// TIA Portal V18 export
ORGANIZATION_BLOCK "00-Alarms"   // OB126, LAD, ProgramCycle
TITLE = Alarms / "Main Program Sweep (Cycle)"
{ S7_Optimized_Access := 'TRUE' }
VERSION : 0.1
// stored: AutoNumber true, IsIECCheckEnabled false, SetENOAutomatically false
   VAR_INPUT
      Initial_Call : Bool;   // Initial call of this OB
      Remanence : Bool;   // =True, if remanent data are available
   END_VAR
BEGIN

REGION Network 1
   // Sınıflandıramadığım Alarm Listesi
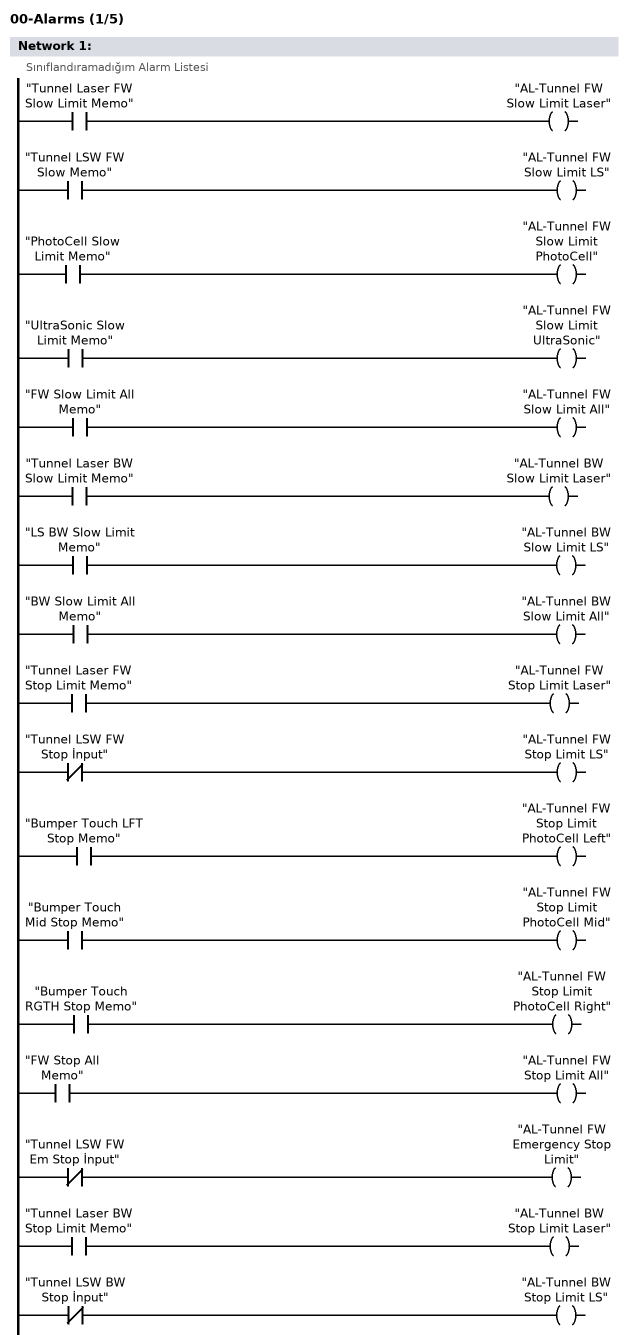
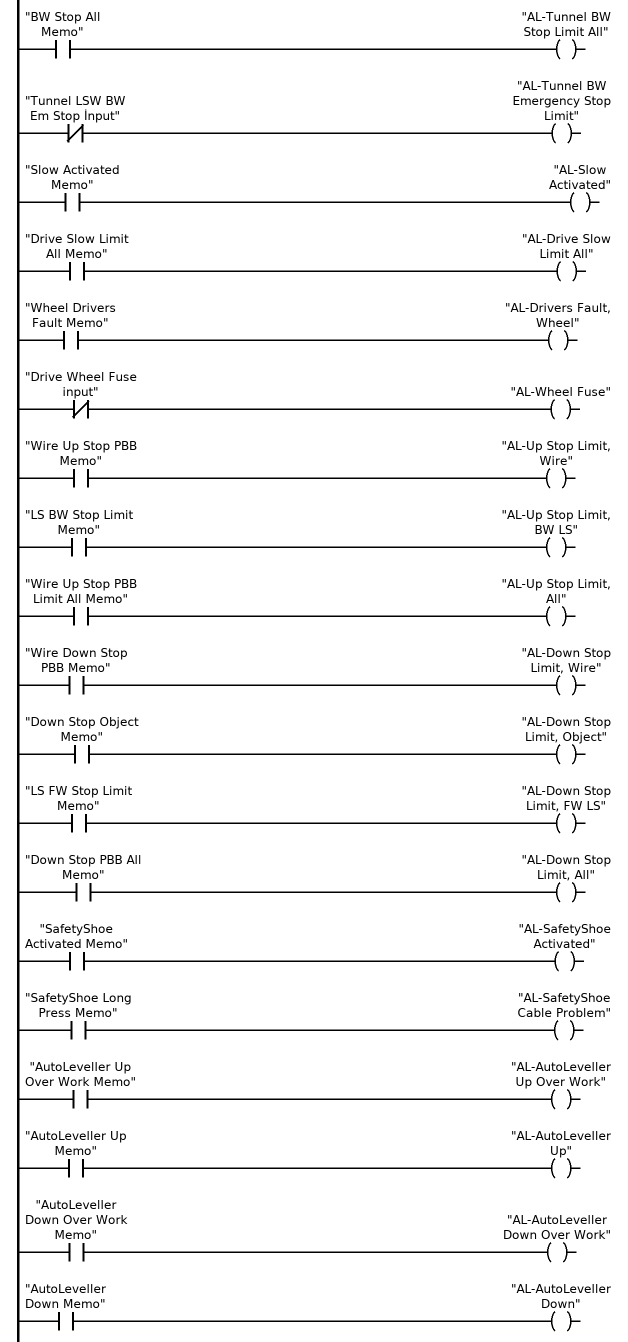
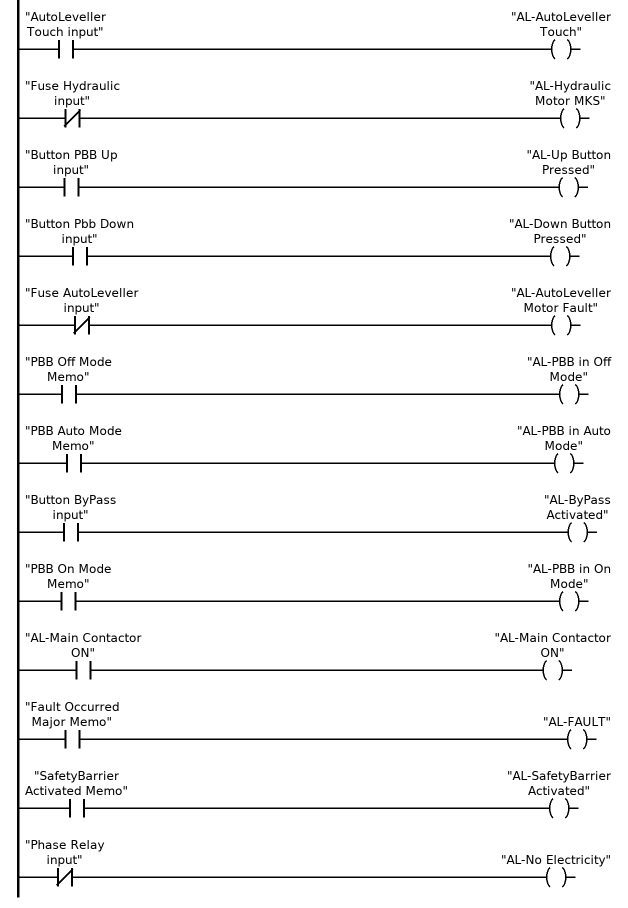
   RUNG wire#powerrail
      Contact( "Tunnel Laser FW Slow Limit Memo" )
      Coil( "AL-Tunnel FW Slow Limit Laser" )
   END_RUNG
   RUNG wire#powerrail
      Contact( "Tunnel LSW FW Slow Memo" )
      Coil( "AL-Tunnel FW Slow Limit LS" )
   END_RUNG
   RUNG wire#powerrail
      Contact( "PhotoCell Slow Limit Memo" )
      Coil( "AL-Tunnel FW Slow Limit PhotoCell" )
   END_RUNG
   RUNG wire#powerrail
      Contact( "UltraSonic Slow Limit Memo" )
      Coil( "AL-Tunnel FW Slow Limit UltraSonic" )
   END_RUNG
   RUNG wire#powerrail
      Contact( "FW Slow Limit All Memo" )
      Coil( "AL-Tunnel FW Slow Limit All" )
   END_RUNG
   RUNG wire#powerrail
      Contact( "Tunnel Laser BW Slow Limit Memo" )
      Coil( "AL-Tunnel BW Slow Limit Laser" )
   END_RUNG
   RUNG wire#powerrail
      Contact( "LS BW Slow Limit Memo" )
      Coil( "AL-Tunnel BW Slow Limit LS" )
   END_RUNG
   RUNG wire#powerrail
      Contact( "BW Slow Limit All Memo" )
      Coil( "AL-Tunnel BW Slow Limit All" )
   END_RUNG
   RUNG wire#powerrail
      Contact( "Tunnel Laser FW Stop Limit Memo" )
      Coil( "AL-Tunnel FW Stop Limit Laser" )
   END_RUNG
   RUNG wire#powerrail
      I_Contact( "Tunnel LSW FW Stop İnput" )
      Coil( "AL-Tunnel FW Stop Limit LS" )
   END_RUNG
   RUNG wire#powerrail
      Contact( "Bumper Touch LFT Stop Memo" )
      Coil( "AL-Tunnel FW Stop Limit PhotoCell Left" )
   END_RUNG
   RUNG wire#powerrail
      Contact( "Bumper Touch Mid Stop Memo" )
      Coil( "AL-Tunnel FW Stop Limit PhotoCell Mid" )
   END_RUNG
   RUNG wire#powerrail
      Contact( "Bumper Touch RGTH Stop Memo" )
      Coil( "AL-Tunnel FW Stop Limit PhotoCell Right" )
   END_RUNG
   RUNG wire#powerrail
      Contact( "FW Stop All Memo" )
      Coil( "AL-Tunnel FW Stop Limit All" )
   END_RUNG
   RUNG wire#powerrail
      I_Contact( "Tunnel LSW FW Em Stop İnput" )
      Coil( "AL-Tunnel FW Emergency Stop Limit" )
   END_RUNG
   RUNG wire#powerrail
      Contact( "Tunnel Laser BW Stop Limit Memo" )
      Coil( "AL-Tunnel BW Stop Limit Laser" )
   END_RUNG
   RUNG wire#powerrail
      I_Contact( "Tunnel LSW BW Stop İnput" )
      Coil( "AL-Tunnel BW Stop Limit LS" )
   END_RUNG
   RUNG wire#powerrail
      Contact( "BW Stop All Memo" )
      Coil( "AL-Tunnel BW Stop Limit All" )
   END_RUNG
   RUNG wire#powerrail
      I_Contact( "Tunnel LSW BW Em Stop İnput" )
      Coil( "AL-Tunnel BW Emergency Stop Limit" )
   END_RUNG
   RUNG wire#powerrail
      Contact( "Slow Activated Memo" )
      Coil( "AL-Slow Activated" )
   END_RUNG
   RUNG wire#powerrail
      Contact( "Drive Slow Limit All Memo" )
      Coil( "AL-Drive Slow Limit All" )
   END_RUNG
   RUNG wire#powerrail
      Contact( "Wheel Drivers Fault Memo" )
      Coil( "AL-Drivers Fault, Wheel" )
   END_RUNG
   RUNG wire#powerrail
      I_Contact( "Drive Wheel Fuse input" )
      Coil( "AL-Wheel Fuse" )
   END_RUNG
   RUNG wire#powerrail
      Contact( "Wire Up Stop PBB Memo" )
      Coil( "AL-Up Stop Limit, Wire" )
   END_RUNG
   RUNG wire#powerrail
      Contact( "LS BW Stop Limit Memo" )
      Coil( "AL-Up Stop Limit, BW LS" )
   END_RUNG
   RUNG wire#powerrail
      Contact( "Wire Up Stop PBB Limit All Memo" )
      Coil( "AL-Up Stop Limit, All" )
   END_RUNG
   RUNG wire#powerrail
      Contact( "Wire Down Stop PBB Memo" )
      Coil( "AL-Down Stop Limit, Wire" )
   END_RUNG
   RUNG wire#powerrail
      Contact( "Down Stop Object Memo" )
      Coil( "AL-Down Stop Limit, Object" )
   END_RUNG
   RUNG wire#powerrail
      Contact( "LS FW Stop Limit Memo" )
      Coil( "AL-Down Stop Limit, FW LS" )
   END_RUNG
   RUNG wire#powerrail
      Contact( "Down Stop PBB All Memo" )
      Coil( "AL-Down Stop Limit, All" )
   END_RUNG
   RUNG wire#powerrail
      Contact( "SafetyShoe Activated Memo" )
      Coil( "AL-SafetyShoe Activated" )
   END_RUNG
   RUNG wire#powerrail
      Contact( "SafetyShoe Long Press Memo" )
      Coil( "AL-SafetyShoe Cable Problem" )
   END_RUNG
   RUNG wire#powerrail
      Contact( "AutoLeveller Up Over Work Memo" )
      Coil( "AL-AutoLeveller Up Over Work" )
   END_RUNG
   RUNG wire#powerrail
      Contact( "AutoLeveller Up Memo" )
      Coil( "AL-AutoLeveller Up" )
   END_RUNG
   RUNG wire#powerrail
      Contact( "AutoLeveller Down Over Work Memo" )
      Coil( "AL-AutoLeveller Down Over Work" )
   END_RUNG
   RUNG wire#powerrail
      Contact( "AutoLeveller Down Memo" )
      Coil( "AL-AutoLeveller Down" )
   END_RUNG
   RUNG wire#powerrail
      Contact( "AutoLeveller Touch input" )
      Coil( "AL-AutoLeveller Touch" )
   END_RUNG
   RUNG wire#powerrail
      I_Contact( "Fuse Hydraulic input" )
      Coil( "AL-Hydraulic Motor MKS" )
   END_RUNG
   RUNG wire#powerrail
      Contact( "Button PBB Up input" )
      Coil( "AL-Up Button Pressed" )
   END_RUNG
   RUNG wire#powerrail
      Contact( "Button Pbb Down input" )
      Coil( "AL-Down Button Pressed" )
   END_RUNG
   RUNG wire#powerrail
      I_Contact( "Fuse AutoLeveller input" )
      Coil( "AL-AutoLeveller Motor Fault" )
   END_RUNG
   RUNG wire#powerrail
      Contact( "PBB Off Mode Memo" )
      Coil( "AL-PBB in Off Mode" )
   END_RUNG
   RUNG wire#powerrail
      Contact( "PBB Auto Mode Memo" )
      Coil( "AL-PBB in Auto Mode" )
   END_RUNG
   RUNG wire#powerrail
      Contact( "Button ByPass input" )
      Coil( "AL-ByPass Activated" )
   END_RUNG
   RUNG wire#powerrail
      Contact( "PBB On Mode Memo" )
      Coil( "AL-PBB in On Mode" )
   END_RUNG
   RUNG wire#powerrail
      Contact( "AL-Main Contactor ON" )
      Coil( "AL-Main Contactor ON" )
   END_RUNG
   RUNG wire#powerrail
      Contact( "Fault Occurred Major Memo" )
      Coil( "AL-FAULT" )
   END_RUNG
   RUNG wire#powerrail
      Contact( "SafetyBarrier Activated Memo" )
      Coil( "AL-SafetyBarrier Activated" )
   END_RUNG
   RUNG wire#powerrail
      I_Contact( "Phase Relay input" )
      Coil( "AL-No Electricity" )
   END_RUNG
   // the same network as SCL:
   "AL-Tunnel FW Slow Limit Laser" := "Tunnel Laser FW Slow Limit Memo";
   "AL-Tunnel FW Slow Limit LS" := "Tunnel LSW FW Slow Memo";
   "AL-Tunnel FW Slow Limit PhotoCell" := "PhotoCell Slow Limit Memo";
   "AL-Tunnel FW Slow Limit UltraSonic" := "UltraSonic Slow Limit Memo";
   "AL-Tunnel FW Slow Limit All" := "FW Slow Limit All Memo";
   "AL-Tunnel BW Slow Limit Laser" := "Tunnel Laser BW Slow Limit Memo";
   "AL-Tunnel BW Slow Limit LS" := "LS BW Slow Limit Memo";
   "AL-Tunnel BW Slow Limit All" := "BW Slow Limit All Memo";
   "AL-Tunnel FW Stop Limit Laser" := "Tunnel Laser FW Stop Limit Memo";
   "AL-Tunnel FW Stop Limit LS" := NOT "Tunnel LSW FW Stop İnput";
   "AL-Tunnel FW Stop Limit PhotoCell Left" := "Bumper Touch LFT Stop Memo";
   "AL-Tunnel FW Stop Limit PhotoCell Mid" := "Bumper Touch Mid Stop Memo";
   "AL-Tunnel FW Stop Limit PhotoCell Right" := "Bumper Touch RGTH Stop Memo";
   "AL-Tunnel FW Stop Limit All" := "FW Stop All Memo";
   "AL-Tunnel FW Emergency Stop Limit" := NOT "Tunnel LSW FW Em Stop İnput";
   "AL-Tunnel BW Stop Limit Laser" := "Tunnel Laser BW Stop Limit Memo";
   "AL-Tunnel BW Stop Limit LS" := NOT "Tunnel LSW BW Stop İnput";
   "AL-Tunnel BW Stop Limit All" := "BW Stop All Memo";
   "AL-Tunnel BW Emergency Stop Limit" := NOT "Tunnel LSW BW Em Stop İnput";
   "AL-Slow Activated" := "Slow Activated Memo";
   "AL-Drive Slow Limit All" := "Drive Slow Limit All Memo";
   "AL-Drivers Fault, Wheel" := "Wheel Drivers Fault Memo";
   "AL-Wheel Fuse" := NOT "Drive Wheel Fuse input";
   "AL-Up Stop Limit, Wire" := "Wire Up Stop PBB Memo";
   "AL-Up Stop Limit, BW LS" := "LS BW Stop Limit Memo";
   "AL-Up Stop Limit, All" := "Wire Up Stop PBB Limit All Memo";
   "AL-Down Stop Limit, Wire" := "Wire Down Stop PBB Memo";
   "AL-Down Stop Limit, Object" := "Down Stop Object Memo";
   "AL-Down Stop Limit, FW LS" := "LS FW Stop Limit Memo";
   "AL-Down Stop Limit, All" := "Down Stop PBB All Memo";
   "AL-SafetyShoe Activated" := "SafetyShoe Activated Memo";
   "AL-SafetyShoe Cable Problem" := "SafetyShoe Long Press Memo";
   "AL-AutoLeveller Up Over Work" := "AutoLeveller Up Over Work Memo";
   "AL-AutoLeveller Up" := "AutoLeveller Up Memo";
   "AL-AutoLeveller Down Over Work" := "AutoLeveller Down Over Work Memo";
   "AL-AutoLeveller Down" := "AutoLeveller Down Memo";
   "AL-AutoLeveller Touch" := "AutoLeveller Touch input";
   "AL-Hydraulic Motor MKS" := NOT "Fuse Hydraulic input";
   "AL-Up Button Pressed" := "Button PBB Up input";
   "AL-Down Button Pressed" := "Button Pbb Down input";
   "AL-AutoLeveller Motor Fault" := NOT "Fuse AutoLeveller input";
   "AL-PBB in Off Mode" := "PBB Off Mode Memo";
   "AL-PBB in Auto Mode" := "PBB Auto Mode Memo";
   "AL-ByPass Activated" := "Button ByPass input";
   "AL-PBB in On Mode" := "PBB On Mode Memo";
   "AL-Main Contactor ON" := "AL-Main Contactor ON";
   "AL-FAULT" := "Fault Occurred Major Memo";
   "AL-SafetyBarrier Activated" := "SafetyBarrier Activated Memo";
   "AL-No Electricity" := NOT "Phase Relay input";
END_REGION

REGION Network 2: Drive
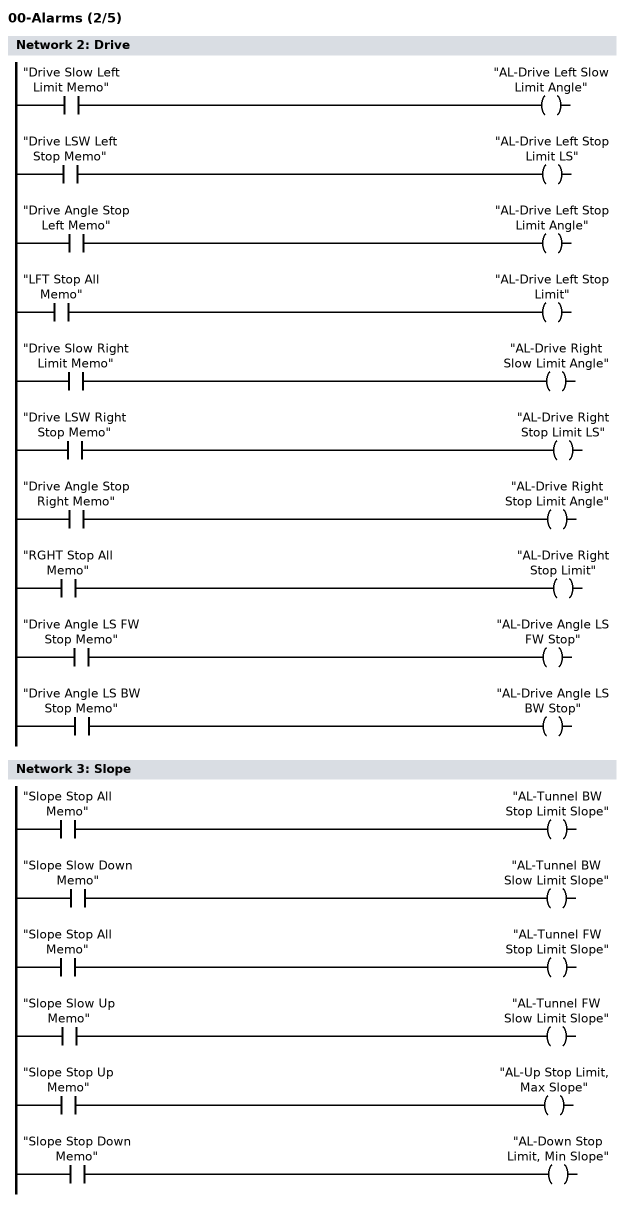
   RUNG wire#powerrail
      Contact( "Drive Slow Left Limit Memo" )
      Coil( "AL-Drive Left Slow Limit Angle" )
   END_RUNG
   RUNG wire#powerrail
      Contact( "Drive LSW Left Stop Memo" )
      Coil( "AL-Drive Left Stop Limit LS" )
   END_RUNG
   RUNG wire#powerrail
      Contact( "Drive Angle Stop Left Memo" )
      Coil( "AL-Drive Left Stop Limit Angle" )
   END_RUNG
   RUNG wire#powerrail
      Contact( "LFT Stop All Memo" )
      Coil( "AL-Drive Left Stop Limit" )
   END_RUNG
   RUNG wire#powerrail
      Contact( "Drive Slow Right Limit Memo" )
      Coil( "AL-Drive Right Slow Limit Angle" )
   END_RUNG
   RUNG wire#powerrail
      Contact( "Drive LSW Right Stop Memo" )
      Coil( "AL-Drive Right Stop Limit LS" )
   END_RUNG
   RUNG wire#powerrail
      Contact( "Drive Angle Stop Right Memo" )
      Coil( "AL-Drive Right Stop Limit Angle" )
   END_RUNG
   RUNG wire#powerrail
      Contact( "RGHT Stop All Memo" )
      Coil( "AL-Drive Right Stop Limit" )
   END_RUNG
   RUNG wire#powerrail
      Contact( "Drive Angle LS FW Stop Memo" )
      Coil( "AL-Drive Angle LS FW Stop" )
   END_RUNG
   RUNG wire#powerrail
      Contact( "Drive Angle LS BW Stop Memo" )
      Coil( "AL-Drive Angle LS BW Stop" )
   END_RUNG
   // the same network as SCL:
   "AL-Drive Left Slow Limit Angle" := "Drive Slow Left Limit Memo";
   "AL-Drive Left Stop Limit LS" := "Drive LSW Left Stop Memo";
   "AL-Drive Left Stop Limit Angle" := "Drive Angle Stop Left Memo";
   "AL-Drive Left Stop Limit" := "LFT Stop All Memo";
   "AL-Drive Right Slow Limit Angle" := "Drive Slow Right Limit Memo";
   "AL-Drive Right Stop Limit LS" := "Drive LSW Right Stop Memo";
   "AL-Drive Right Stop Limit Angle" := "Drive Angle Stop Right Memo";
   "AL-Drive Right Stop Limit" := "RGHT Stop All Memo";
   "AL-Drive Angle LS FW Stop" := "Drive Angle LS FW Stop Memo";
   "AL-Drive Angle LS BW Stop" := "Drive Angle LS BW Stop Memo";
END_REGION

REGION Network 3: Slope
   RUNG wire#powerrail
      Contact( "Slope Stop All Memo" )
      Coil( "AL-Tunnel BW Stop Limit Slope" )
   END_RUNG
   RUNG wire#powerrail
      Contact( "Slope Slow Down Memo" )
      Coil( "AL-Tunnel BW Slow Limit Slope" )
   END_RUNG
   RUNG wire#powerrail
      Contact( "Slope Stop All Memo" )
      Coil( "AL-Tunnel FW Stop Limit Slope" )
   END_RUNG
   RUNG wire#powerrail
      Contact( "Slope Slow Up Memo" )
      Coil( "AL-Tunnel FW Slow Limit Slope" )
   END_RUNG
   RUNG wire#powerrail
      Contact( "Slope Stop Up Memo" )
      Coil( "AL-Up Stop Limit, Max Slope" )
   END_RUNG
   RUNG wire#powerrail
      Contact( "Slope Stop Down Memo" )
      Coil( "AL-Down Stop Limit, Min Slope" )
   END_RUNG
   // the same network as SCL:
   "AL-Tunnel BW Stop Limit Slope" := "Slope Stop All Memo";
   "AL-Tunnel BW Slow Limit Slope" := "Slope Slow Down Memo";
   "AL-Tunnel FW Stop Limit Slope" := "Slope Stop All Memo";
   "AL-Tunnel FW Slow Limit Slope" := "Slope Slow Up Memo";
   "AL-Up Stop Limit, Max Slope" := "Slope Stop Up Memo";
   "AL-Down Stop Limit, Min Slope" := "Slope Stop Down Memo";
END_REGION

REGION Network 4: Rotunda
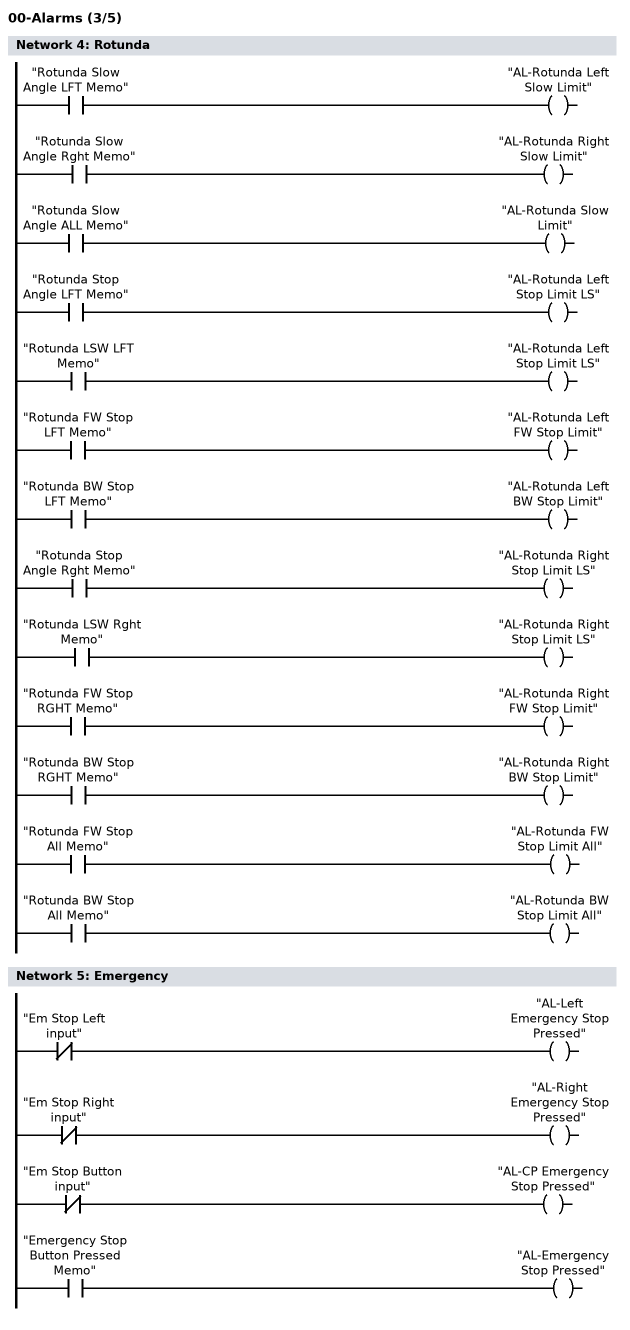
   RUNG wire#powerrail
      Contact( "Rotunda Slow Angle LFT Memo" )
      Coil( "AL-Rotunda Left Slow Limit" )
   END_RUNG
   RUNG wire#powerrail
      Contact( "Rotunda Slow Angle Rght Memo" )
      Coil( "AL-Rotunda Right Slow Limit" )
   END_RUNG
   RUNG wire#powerrail
      Contact( "Rotunda Slow Angle ALL Memo" )
      Coil( "AL-Rotunda Slow Limit" )
   END_RUNG
   RUNG wire#powerrail
      Contact( "Rotunda Stop Angle LFT Memo" )
      Coil( "AL-Rotunda Left Stop Limit LS" )
   END_RUNG
   RUNG wire#powerrail
      Contact( "Rotunda LSW LFT Memo" )
      Coil( "AL-Rotunda Left Stop Limit LS" )
   END_RUNG
   RUNG wire#powerrail
      Contact( "Rotunda FW Stop LFT Memo" )
      Coil( "AL-Rotunda Left FW Stop Limit" )
   END_RUNG
   RUNG wire#powerrail
      Contact( "Rotunda BW Stop LFT Memo" )
      Coil( "AL-Rotunda Left BW Stop Limit" )
   END_RUNG
   RUNG wire#powerrail
      Contact( "Rotunda Stop Angle Rght Memo" )
      Coil( "AL-Rotunda Right Stop Limit LS" )
   END_RUNG
   RUNG wire#powerrail
      Contact( "Rotunda LSW Rght Memo" )
      Coil( "AL-Rotunda Right Stop Limit LS" )
   END_RUNG
   RUNG wire#powerrail
      Contact( "Rotunda FW Stop RGHT Memo" )
      Coil( "AL-Rotunda Right FW Stop Limit" )
   END_RUNG
   RUNG wire#powerrail
      Contact( "Rotunda BW Stop RGHT Memo" )
      Coil( "AL-Rotunda Right BW Stop Limit" )
   END_RUNG
   RUNG wire#powerrail
      Contact( "Rotunda FW Stop All Memo" )
      Coil( "AL-Rotunda FW Stop Limit All" )
   END_RUNG
   RUNG wire#powerrail
      Contact( "Rotunda BW Stop All Memo" )
      Coil( "AL-Rotunda BW Stop Limit All" )
   END_RUNG
   // the same network as SCL:
   "AL-Rotunda Left Slow Limit" := "Rotunda Slow Angle LFT Memo";
   "AL-Rotunda Right Slow Limit" := "Rotunda Slow Angle Rght Memo";
   "AL-Rotunda Slow Limit" := "Rotunda Slow Angle ALL Memo";
   "AL-Rotunda Left Stop Limit LS" := "Rotunda Stop Angle LFT Memo";
   "AL-Rotunda Left Stop Limit LS" := "Rotunda LSW LFT Memo";
   "AL-Rotunda Left FW Stop Limit" := "Rotunda FW Stop LFT Memo";
   "AL-Rotunda Left BW Stop Limit" := "Rotunda BW Stop LFT Memo";
   "AL-Rotunda Right Stop Limit LS" := "Rotunda Stop Angle Rght Memo";
   "AL-Rotunda Right Stop Limit LS" := "Rotunda LSW Rght Memo";
   "AL-Rotunda Right FW Stop Limit" := "Rotunda FW Stop RGHT Memo";
   "AL-Rotunda Right BW Stop Limit" := "Rotunda BW Stop RGHT Memo";
   "AL-Rotunda FW Stop Limit All" := "Rotunda FW Stop All Memo";
   "AL-Rotunda BW Stop Limit All" := "Rotunda BW Stop All Memo";
END_REGION

REGION Network 5: Emergency
   RUNG wire#powerrail
      I_Contact( "Em Stop Left input" )
      Coil( "AL-Left Emergency Stop Pressed" )
   END_RUNG
   RUNG wire#powerrail
      I_Contact( "Em Stop Right input" )
      Coil( "AL-Right Emergency Stop Pressed" )
   END_RUNG
   RUNG wire#powerrail
      I_Contact( "Em Stop Button input" )
      Coil( "AL-CP Emergency Stop Pressed" )
   END_RUNG
   RUNG wire#powerrail
      Contact( "Emergency Stop Button Pressed Memo" )
      Coil( "AL-Emergency Stop Pressed" )
   END_RUNG
   // the same network as SCL:
   "AL-Left Emergency Stop Pressed" := NOT "Em Stop Left input";
   "AL-Right Emergency Stop Pressed" := NOT "Em Stop Right input";
   "AL-CP Emergency Stop Pressed" := NOT "Em Stop Button input";
   "AL-Emergency Stop Pressed" := "Emergency Stop Button Pressed Memo";
END_REGION

REGION Network 6: Cab
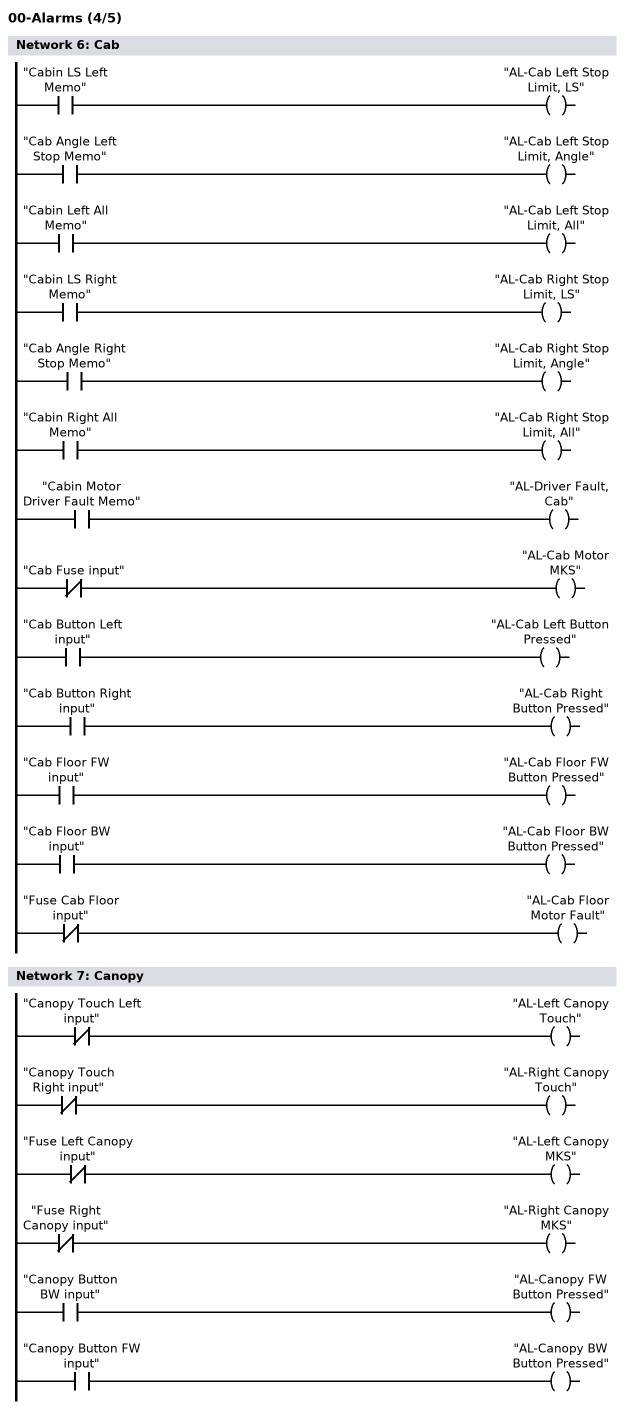
   RUNG wire#powerrail
      Contact( "Cabin LS Left Memo" )
      Coil( "AL-Cab Left Stop Limit, LS" )
   END_RUNG
   RUNG wire#powerrail
      Contact( "Cab Angle Left Stop Memo" )
      Coil( "AL-Cab Left Stop Limit, Angle" )
   END_RUNG
   RUNG wire#powerrail
      Contact( "Cabin Left All Memo" )
      Coil( "AL-Cab Left Stop Limit, All" )
   END_RUNG
   RUNG wire#powerrail
      Contact( "Cabin LS Right Memo" )
      Coil( "AL-Cab Right Stop Limit, LS" )
   END_RUNG
   RUNG wire#powerrail
      Contact( "Cab Angle Right Stop Memo" )
      Coil( "AL-Cab Right Stop Limit, Angle" )
   END_RUNG
   RUNG wire#powerrail
      Contact( "Cabin Right All Memo" )
      Coil( "AL-Cab Right Stop Limit, All" )
   END_RUNG
   RUNG wire#powerrail
      Contact( "Cabin Motor Driver Fault Memo" )
      Coil( "AL-Driver Fault, Cab" )
   END_RUNG
   RUNG wire#powerrail
      I_Contact( "Cab Fuse input" )
      Coil( "AL-Cab Motor MKS" )
   END_RUNG
   RUNG wire#powerrail
      Contact( "Cab Button Left input" )
      Coil( "AL-Cab Left Button Pressed" )
   END_RUNG
   RUNG wire#powerrail
      Contact( "Cab Button Right input" )
      Coil( "AL-Cab Right Button Pressed" )
   END_RUNG
   RUNG wire#powerrail
      Contact( "Cab Floor FW input" )
      Coil( "AL-Cab Floor FW Button Pressed" )
   END_RUNG
   RUNG wire#powerrail
      Contact( "Cab Floor BW input" )
      Coil( "AL-Cab Floor BW Button Pressed" )
   END_RUNG
   RUNG wire#powerrail
      I_Contact( "Fuse Cab Floor input" )
      Coil( "AL-Cab Floor Motor Fault" )
   END_RUNG
   // the same network as SCL:
   "AL-Cab Left Stop Limit, LS" := "Cabin LS Left Memo";
   "AL-Cab Left Stop Limit, Angle" := "Cab Angle Left Stop Memo";
   "AL-Cab Left Stop Limit, All" := "Cabin Left All Memo";
   "AL-Cab Right Stop Limit, LS" := "Cabin LS Right Memo";
   "AL-Cab Right Stop Limit, Angle" := "Cab Angle Right Stop Memo";
   "AL-Cab Right Stop Limit, All" := "Cabin Right All Memo";
   "AL-Driver Fault, Cab" := "Cabin Motor Driver Fault Memo";
   "AL-Cab Motor MKS" := NOT "Cab Fuse input";
   "AL-Cab Left Button Pressed" := "Cab Button Left input";
   "AL-Cab Right Button Pressed" := "Cab Button Right input";
   "AL-Cab Floor FW Button Pressed" := "Cab Floor FW input";
   "AL-Cab Floor BW Button Pressed" := "Cab Floor BW input";
   "AL-Cab Floor Motor Fault" := NOT "Fuse Cab Floor input";
END_REGION

REGION Network 7: Canopy
   RUNG wire#powerrail
      I_Contact( "Canopy Touch Left input" )
      Coil( "AL-Left Canopy Touch" )
   END_RUNG
   RUNG wire#powerrail
      I_Contact( "Canopy Touch Right input" )
      Coil( "AL-Right Canopy Touch" )
   END_RUNG
   RUNG wire#powerrail
      I_Contact( "Fuse Left Canopy input" )
      Coil( "AL-Left Canopy MKS" )
   END_RUNG
   RUNG wire#powerrail
      I_Contact( "Fuse Right Canopy input" )
      Coil( "AL-Right Canopy MKS" )
   END_RUNG
   RUNG wire#powerrail
      Contact( "Canopy Button BW input" )
      Coil( "AL-Canopy FW Button Pressed" )
   END_RUNG
   RUNG wire#powerrail
      Contact( "Canopy Button FW input" )
      Coil( "AL-Canopy BW Button Pressed" )
   END_RUNG
   // the same network as SCL:
   "AL-Left Canopy Touch" := NOT "Canopy Touch Left input";
   "AL-Right Canopy Touch" := NOT "Canopy Touch Right input";
   "AL-Left Canopy MKS" := NOT "Fuse Left Canopy input";
   "AL-Right Canopy MKS" := NOT "Fuse Right Canopy input";
   "AL-Canopy FW Button Pressed" := "Canopy Button BW input";
   "AL-Canopy BW Button Pressed" := "Canopy Button FW input";
END_REGION

REGION Network 8: PCA and GPU Service
END_REGION

REGION Network 9: Services
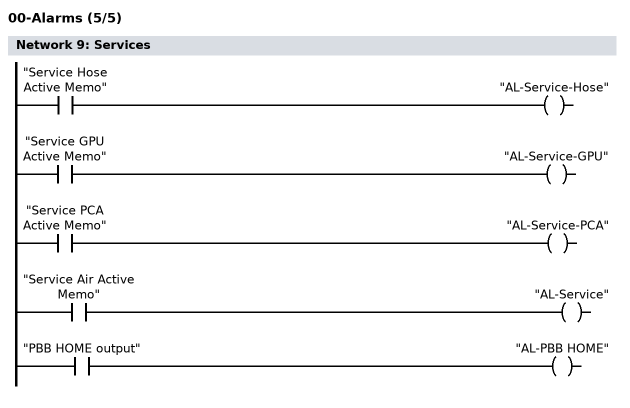
   RUNG wire#powerrail
      Contact( "Service Hose Active Memo" )
      Coil( "AL-Service-Hose" )
   END_RUNG
   RUNG wire#powerrail
      Contact( "Service GPU Active Memo" )
      Coil( "AL-Service-GPU" )
   END_RUNG
   RUNG wire#powerrail
      Contact( "Service PCA Active Memo" )
      Coil( "AL-Service-PCA" )
   END_RUNG
   RUNG wire#powerrail
      Contact( "Service Air Active Memo" )
      Coil( "AL-Service" )
   END_RUNG
   RUNG wire#powerrail
      Contact( "PBB HOME output" )
      Coil( "AL-PBB HOME" )
   END_RUNG
   // the same network as SCL:
   "AL-Service-Hose" := "Service Hose Active Memo";
   "AL-Service-GPU" := "Service GPU Active Memo";
   "AL-Service-PCA" := "Service PCA Active Memo";
   "AL-Service" := "Service Air Active Memo";
   "AL-PBB HOME" := "PBB HOME output";
END_REGION
END_ORGANIZATION_BLOCK
